ABB RAPID module: HSLU_Data.modx

MODULE HSLU_Data

    !************************************************
    ! Declaration :     string
    !************************************************
    !
    TASK PERS string st_HSLU_Header:="Swissbau";

    !************************************************
    ! Declaration :     num
    !************************************************
    !
    TASK PERS num n_HSLU_ActOverride:=0;
    CONST robtarget Nullpunkt := [[0,0,0],[0.0983481,0.372237,0.922828,0.012505],[-1,-1,1,0],[9E+09,9E+09,9E+09,9E+09,9E+09,9E+09]];

ENDMODULE
